PROGRAM P30_ManualControl
VAR
	i 	: INT;
	
	Temp_1_Ramping:ARRAY[1..6]OF  INT;
	Temp_1_target: ARRAY[1..6]OF  INT;
	Temp_1_BufferTarget: ARRAY[1..6]OF  INT;
	
	fbAnalogDeviceRampControl:FB_AnalogDeviceRampControl;
	

END_VAR

fbAnalogDeviceRampControl();

END_PROGRAM

(* stored: Version 1.1.0.1
   POU P30_ManualControl: Id {98ee4f4f-99e9-426e-9dfa-55ddf51d552b}, SpecialFunc None *)
